METHOD _copyToModel_SM_ThermoVac
  VAR_IN_OUT
    {attribute 'OPC.UA.DA' := '0'}
    model : M_SM_ThermoVac;
  END_VAR
                  model.editableConfig := THIS^.editableConfig;
model.actualStatus := THIS^.actualStatus;
model.config := THIS^.config;
model.stat := THIS^.stat;
THIS^.parts.thermo._copyToModel_Thermo( model := model.parts.thermo );
THIS^.parts.vac._copyToModel_Vac( model := model.parts.vac );
THIS^.parts.configManager._copyToModel_ConfigManager( model := model.parts.configManager );
THIS^.proc.initialize._copyToModel_Process( model := model.proc.initialize );
THIS^.proc.reset._copyToModel_Process( model := model.proc.reset );
THIS^.proc.lock._copyToModel_Process( model := model.proc.lock );
THIS^.proc.unlock._copyToModel_Process( model := model.proc.unlock );

                
END_METHOD
END_FUNCTION_BLOCK

FUNCTION_BLOCK ForceHeater EXTENDS BaseProcess
  VAR_INPUT
    {attribute 'OPC.UA.DA' := '1'}
    {attribute 'OPC.UA.DA.Access' := '3'}
    {attribute 'TcHmiSymbol.Show'}
    set : ForceHeaterArgs;  (* Arguments to be set, before writing do_request TRUE *)
  END_VAR
  VAR_OUTPUT
    {attribute 'OPC.UA.DA' := '0'}
    get : ForceHeaterArgs;  (* Arguments in use by the process, if do_request was accepted *)
  END_VAR

            IF do_request THEN
    do_request_result := request( power := set.power );
    do_request := FALSE;
END_IF;
SUPER^();

          

{attribute 'TcRpcEnable' := '1'}
METHOD start
  VAR_INPUT
    power : REAL;
  END_VAR
                  THIS^.get.power := power;
THIS^.stat.busy := BusyStatus.busy;
THIS^.stat.health := HealthStatus.good;

                
END_METHOD

{attribute 'TcRpcEnable' := '1'}
METHOD request : RequestResults
  VAR_INPUT
    power : REAL;
  END_VAR
                  IF THIS^.stat.enabled = EnabledStatus.enabled THEN
    request := RequestResults.ACCEPTED;
    THIS^.start( power := power );
ELSE
    request := RequestResults.REJECTED;
END_IF;

                
END_METHOD

METHOD _copyFromModel_ForceHeater
  VAR_IN_OUT
    {attribute 'OPC.UA.DA' := '0'}
    model : M_ForceHeater;
  END_VAR
                  THIS^.set := model.set;
SUPER^._copyFromModel_BaseProcess( model := model );

                
END_METHOD

METHOD _copyToModel_ForceHeater
  VAR_IN_OUT
    {attribute 'OPC.UA.DA' := '0'}
    model : M_ForceHeater;
  END_VAR
                  model.set := THIS^.set;
SUPER^._copyToModel_BaseProcess( model := model );

                
END_METHOD
END_FUNCTION_BLOCK
